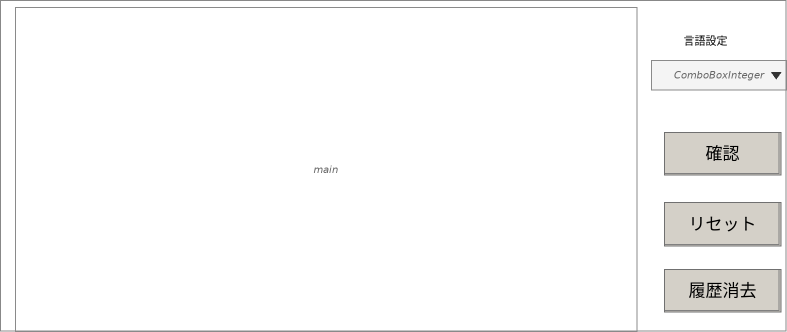
VISUALIZATION Visualization  // 787x332
    Button (664,132 117x43), "確認", colour toggle: AlarmManager.status_unconfirm
        tap AlarmManager.confirm_button_input
    Button (664,202 117x44), "リセット", colour toggle: AlarmManager.status_resetable
        tap AlarmManager.reset_button_input
    TabControl (15,7 622x325)
        shows main()
        shows current()
        shows history()
        [0]: TabTitle=メイン
        [1]: TabTitle=現在アラーム一覧
        [2]: TabTitle=アラーム操作履歴
    Label (664,24 83x34), "言語設定"
    ComboBoxInteger (651,60 136x30), variable: AlarmManager.lang_select_options, text list: 'languages'
    Button (664,269 117x43), "履歴消去"
        tap AlarmManager.history_clear_button_input
END_VISUALIZATION

(* stored: Version 1.1.0.1
   Visu Visualization: Id {230483c7-8b30-4964-94b1-66195911bb3b} *)
